// Mitsubishi GX Works2 project: 시퀀스 전체 반복 회로 예제 (카운터)   PLC: Q03UDV

PROGRAM MAIN
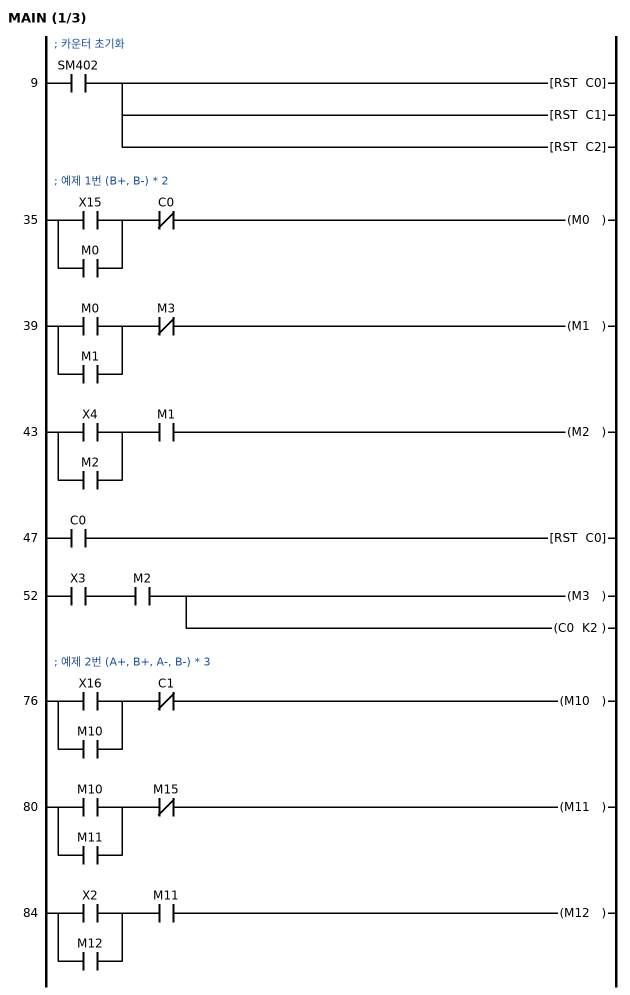
; 카운터 초기화
9     LD      SM402
      RST     C0
      RST     C1
      RST     C2
; 예제 1번 (B+, B-) * 2
35    LD      X15
      OR      M0
      ANI     C0
      OUT     M0
39    LD      M0
      OR      M1
      ANI     M3
      OUT     M1
43    LD      X4
      OR      M2
      AND     M1
      OUT     M2
47    LD      C0
      RST     C0
52    LD      X3
      AND     M2
      OUT     M3
      OUT     C0 K2
; 예제 2번 (A+, B+, A-, B-) * 3
76    LD      X16
      OR      M10
      ANI     C1
      OUT     M10
80    LD      M10
      OR      M11
      ANI     M15
      OUT     M11
84    LD      X2
      OR      M12
      AND     M11
      OUT     M12
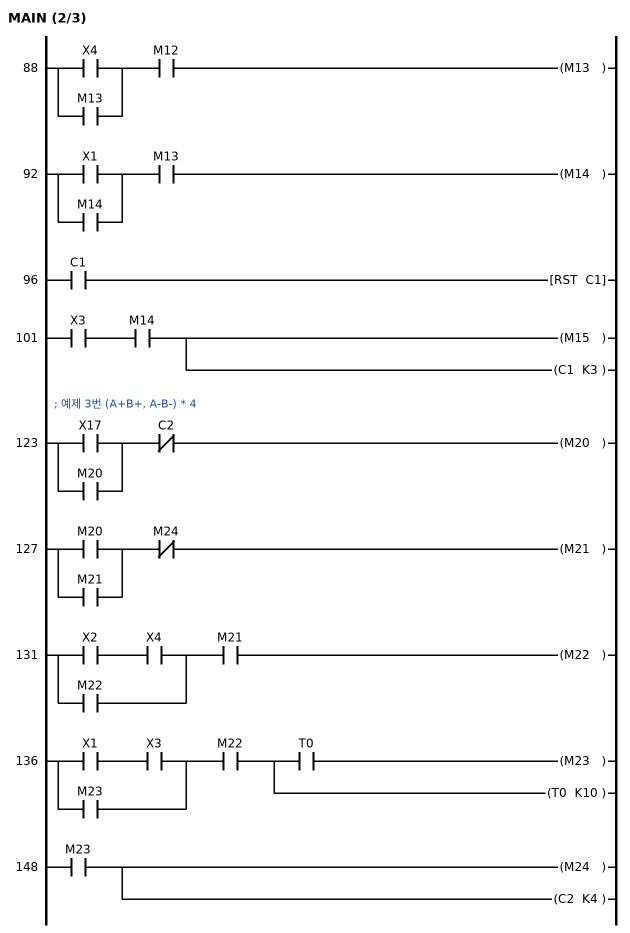
88    LD      X4
      OR      M13
      AND     M12
      OUT     M13
92    LD      X1
      OR      M14
      AND     M13
      OUT     M14
96    LD      C1
      RST     C1
101   LD      X3
      AND     M14
      OUT     M15
      OUT     C1 K3
; 예제 3번 (A+B+, A-B-) * 4
123   LD      X17
      OR      M20
      ANI     C2
      OUT     M20
127   LD      M20
      OR      M21
      ANI     M24
      OUT     M21
131   LD      X2
      AND     X4
      OR      M22
      AND     M21
      OUT     M22
136   LD      X1
      AND     X3
      OR      M23
      AND     M22
      MPS
      AND     T0
      OUT     M23
      MPP
      OUT     T0 K10
148   LD      M23
      OUT     M24
      OUT     C2 K4
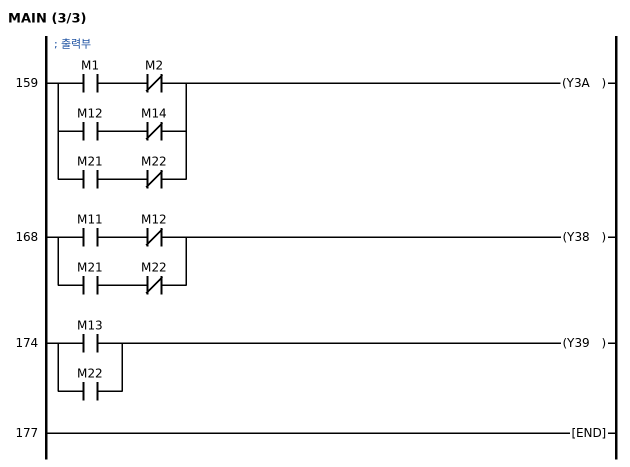
; 출력부
159   LD      M1
      ANI     M2
      LD      M12
      ANI     M14
      ORB
      LD      M21
      ANI     M22
      ORB
      OUT     Y3A
168   LD      M11
      ANI     M12
      LD      M21
      ANI     M22
      ORB
      OUT     Y38
174   LD      M13
      OR      M22
      OUT     Y39
177   END
END_PROGRAM
